FUNCTION F_Message : ST_Message
VAR_INPUT
	eMessage : E_MessageList;
	eFromPeer : E_PeersList;
	eToPeer : E_PeersList;
END_VAR
VAR
END_VAR

F_Message.eMessage := eMessage;
F_Message.eFromPeer := eFromPeer;
F_Message.eToPeer := eToPeer;

END_FUNCTION

(* stored: Version 1.1.0.1, ProductVersion 3.1.4022.16
   POU F_Message: Id {ec0e6791-e369-4a98-a9a5-8239f1aa4efc}, SpecialFunc None *)
